Fanuc KAREL source: ka00092.KL

-- PROVISIONAL review KL for V1013-1; original PC SHA256 facc7f057ce47404d9085bf5c07f4db551ff4f6c0790802104100222673f04e9
-- Incomplete behavior may be omitted. Consult companion uncertainty JSON. Do not deploy.
PROGRAM KA00092
%NOLOCKGROUP
-- UNRESOLVED_DECL SRC type=000199
-- UNRESOLVED_DECL DST type=000199
BEGIN
  -- UNRESOLVED_PC offsets 5-20; opcodes 49,4A
  -- UNRESOLVED_PC offsets 25-29; opcodes 7F
END KA00092
